Yaskawa INFORM job: WELDING-CMF100-ST1-BACK.JBI

/JOB
//NAME WELDING-CMF100-ST1-BACK
//POS
///NPOS 18,18,18,1,0,0
///TOOL 0
///POSTYPE PULSE
///PULSE
C00000=-72547,-33316,-23472,62404,52759,9166
C00001=-66202,-36123,-35615,73106,53931,1994
C00002=-81874,-570,-30266,124582,55821,-26550
C00003=-81654,24349,-54365,147909,11334,-39909
C00004=-81654,24272,-54345,147905,11384,-39900
C00005=-81830,23968,-54649,148018,11360,-39948
C00006=-83267,456,-20171,106212,63641,-16570
C00007=-83261,443,-20218,106265,63625,-16601
C00008=-83230,374,-20246,106195,63616,-16562
C00009=-83229,487,-20120,106130,63627,-16521
C00010=-86542,13642,10788,35301,60758,23207
C00011=-91190,51720,70796,9622,31474,36987
C00012=-100192,52073,75133,2888,27203,40983
C00013=-100192,52073,75133,2888,27203,40983
C00014=-100539,61988,89583,2549,22726,41268
C00015=-84075,-5263,-2872,43968,61349,18923
C00016=-107393,-41599,-17479,-358,59819,45324
C00017=-119865,-4533,-4485,-12604,43978,51654
BC00000=82159
BC00001=82159
BC00002=82159
BC00003=82159
BC00004=82159
BC00005=82159
BC00006=82159
BC00007=82159
BC00008=82159
BC00009=82159
BC00010=82159
BC00011=82159
BC00012=104718
BC00013=104718
BC00014=104718
BC00015=88319
BC00016=88319
BC00017=88861
EC00000=2040211
EC00001=2047981
EC00002=2055875
EC00003=2360213
EC00004=2360213
EC00005=2360213
EC00006=2048000
EC00007=1024000
EC00008=0
EC00009=-1024000
EC00010=-1345219
EC00011=-1515919
EC00012=-1521724
EC00013=-1521724
EC00014=-1521724
EC00015=-1031098
EC00016=-1031098
EC00017=-1003440
///USER 10
///POSTYPE USER
///RECTAN
///RCONF 0,0,0,0,0,0,0,0,0,0,0,0,0,0,0,0,0,0,0,0,0,0,0,0
P00049=2.600,0.000,0.000,0.0000,0.0000,0.0000
//INST
///DATE 2018/10/04 12:06
///ATTR SC,RW
///GROUP1 RB1,BS1
///GROUP2 ST1
NOP
'***** welding station 1 front
MOVJ C00000 BC00000 VJ=25.00  +MOVJ EC00000 VJ=100.00
'***** go to start pos
SMOVL C00001 BC00001 V=166.7 PL=0  +MOVJ EC00001
SFTON P049 UF#(10)
SMOVL C00002 BC00002 V=83.3  +MOVJ EC00002
SMOVC C00003 BC00003 V=83.3 PL=0  +MOVJ EC00003  //start welding
DOUT OT#(656) OFF
TIMER T=0.50
DOUT OT#(656) ON
DOUT OT#(46) ON
DOUT OT#(47) ON
DOUT OT#(45) OFF
MACRO1 MJ#(5) ARGF2
SREFP 1 C00004 BC00004  +REFP EC00004
SREFP 2 C00005 BC00005  +REFP EC00005
ARCON ASF#(1)
SWVON WEV#(1)
SMOVC C00006 BC00006 V=I000  +MOVJ EC00006
SMOVC C00007 BC00007 V=I000  +MOVJ EC00007
SMOVC C00008 BC00008 V=I000  +MOVJ EC00008
SMOVC C00009 BC00009 V=I000  +MOVJ EC00009
SMOVC C00010 BC00010 V=I000  +MOVJ EC00010
SMOVC C00011 BC00011 V=I000  +MOVJ EC00011
SMOVL C00012 BC00012 V=I000  +MOVJ EC00012
ARCOF
SMOVL C00013 BC00013 V=I000  +MOVJ EC00013
MACRO1 MJ#(5) ARGF10
DOUT OT#(656) OFF
SWVOF
TIMER T=5.00
'***** go to end position
SFTOF
SMOVL C00014 BC00014 V=16.7 PL=0  +MOVJ EC00014
SMOVL C00015 BC00015 V=83.3  +MOVJ EC00015
SMOVL C00016 BC00016 V=250.0  +MOVJ EC00016
MOVL C00017 BC00017 V=166.7  +MOVJ EC00017 VJ=100.00
END
